; move to the rack
TRIGGER WHEN DISTANCE=1 DELAY=-1 DO Schrittmerker_R1Place(10880,10501,FPlace_R1_L8_S4_VP1,XPlace_R1_L8_S4_VP1) PRIO=-1
;FOLD PTP Place_R1_L8_S4_VP1 CONT Vel=12 % PPlace_R1_L8_S4_VP1 Tool[1]:Upper Gripper Base[0];%{PE}%R8.3.21,%MKUKATPBASIS,%CMOVE,%VPTP,%P 1:PTP, 2:Place_R1_L8_S4_VP1, 3:C_DIS, 5:12, 7:PPlace_R1_L8_S4_VP1
$BWDSTART=FALSE
PDAT_ACT= PPPlace_R1_L8_S4_VP1
FDAT_ACT= FPlace_R1_L8_S4_VP1
BAS(#PTP_PARAMS,12)
PTP XPlace_R1_L8_S4_VP1 C_DIS
;ENDFOLD
TRIGGER WHEN DISTANCE=1 DELAY=-1 DO Schrittmerker_R1Place(10881,10880,FPlace_R1_L8_S4_VP2,XPlace_R1_L8_S4_VP2) PRIO=-1
;FOLD PTP Place_R1_L8_S4_VP2 CONT Vel=12 % PPlace_R1_L8_S4_VP2 Tool[1]:Upper Gripper Base[0];%{PE}%R8.3.21,%MKUKATPBASIS,%CMOVE,%VPTP,%P 1:PTP, 2:Place_R1_L8_S4_VP2, 3:C_DIS, 5:12, 7:PPlace_R1_L8_S4_VP2
$BWDSTART=FALSE
PDAT_ACT= PPPlace_R1_L8_S4_VP2
FDAT_ACT= FPlace_R1_L8_S4_VP2
BAS(#PTP_PARAMS,12)
PTP XPlace_R1_L8_S4_VP2 C_DIS
;ENDFOLD
TRIGGER WHEN DISTANCE=1 DELAY=-1 DO Schrittmerker_R1Place(10882,10881,FPlace_R1_L8_S4_VP3,XPlace_R1_L8_S4_VP3) PRIO=-1
;FOLD PTP Place_R1_L8_S4_VP3 CONT Vel=12 % PPlace_R1_L8_S4_VP3 Tool[1]:Upper Gripper Base[0];%{PE}%R8.3.21,%MKUKATPBASIS,%CMOVE,%VPTP,%P 1:PTP, 2:Place_R1_L8_S4_VP3, 3:C_DIS, 5:12, 7:PPlace_R1_L8_S4_VP3
$BWDSTART=FALSE
PDAT_ACT= PPPlace_R1_L8_S4_VP3
FDAT_ACT= FPlace_R1_L8_S4_VP3
BAS(#PTP_PARAMS,12)
PTP XPlace_R1_L8_S4_VP3 C_DIS
;ENDFOLD
TRIGGER WHEN DISTANCE=1 DELAY=-1 DO Schrittmerker_R1Place(10883,10882,FPlace_R1_L8_S4_VP4,XPlace_R1_L8_S4_VP4) PRIO=-1
;FOLD PTP Place_R1_L8_S4_VP4 CONT Vel=12 % PPlace_R1_L8_S4_VP4 Tool[1]:Upper Gripper Base[0];%{PE}%R8.3.21,%MKUKATPBASIS,%CMOVE,%VPTP,%P 1:PTP, 2:Place_R1_L8_S4_VP4, 3:C_DIS, 5:12, 7:PPlace_R1_L8_S4_VP4
$BWDSTART=FALSE
PDAT_ACT= PPPlace_R1_L8_S4_VP4
FDAT_ACT= FPlace_R1_L8_S4_VP4
BAS(#PTP_PARAMS,12)
PTP XPlace_R1_L8_S4_VP4 C_DIS
;ENDFOLD
TRIGGER WHEN DISTANCE=1 DELAY=-1 DO Schrittmerker_R1Place(10884,10883,FPlace_R1_L8_S4_VP5,XPlace_R1_L8_S4_VP5) PRIO=-1
;FOLD PTP Place_R1_L8_S4_VP5 CONT Vel=12 % PPlace_R1_L8_S4_VP5 Tool[1]:Upper Gripper Base[0];%{PE}%R8.3.21,%MKUKATPBASIS,%CMOVE,%VPTP,%P 1:PTP, 2:Place_R1_L8_S4_VP5, 3:C_DIS, 5:12, 7:PPlace_R1_L8_S4_VP5
$BWDSTART=FALSE
PDAT_ACT= PPPlace_R1_L8_S4_VP5
FDAT_ACT= FPlace_R1_L8_S4_VP5
BAS(#PTP_PARAMS,12)
PTP XPlace_R1_L8_S4_VP5 C_DIS
;ENDFOLD

TRIGGER WHEN DISTANCE=1 DELAY=-1 DO Schrittmerker_R1Place(10885,10884,FPlace_R1_L8_S4_Check,XPlace_R1_L8_S4_Check) PRIO=-1
;FOLD PTP Place_R1_L8_S4_Check Vel=12 % PPlace_R1_L8_S4_Check Tool[1]:Upper Gripper Base[1]:Rack1;%{PE}%R8.3.21,%MKUKATPBASIS,%CMOVE,%VPTP,%P 1:PTP, 2:Place_R1_L8_S4_Check, 3:, 5:12, 7:PPlace_R1_L8_S4_Check
$BWDSTART=FALSE
PDAT_ACT= PPPlace_R1_L8_S4_Check
FDAT_ACT= FPlace_R1_L8_S4_Check
BAS(#PTP_PARAMS,12)
PTP XPlace_R1_L8_S4_Check
;ENDFOLD

;***************************************************
;FOLD Pruefe Platz frei
IF (DetectPart(CHECK_SHELF,PLACE)==OCCUPIED) THEN
  UP_Rueckzug_R1Place( )
  RETURN
ENDIF
;ENDFOLD
;***************************************************

TRIGGER WHEN DISTANCE=1 DELAY=-1 DO Schrittmerker_R1Place(10886,10885,FPlace_R1_L8_S4_VP6,XPlace_R1_L8_S4_VP6) PRIO=-1
;FOLD LIN Place_R1_L8_S4_VP6 CONT Vel=0.5 m/s LPlace_R1_L8_S4_VP6 Tool[1]:Upper Gripper Base[1]:Rack1;%{PE}%R8.3.21,%MKUKATPBASIS,%CMOVE,%VLIN,%P 1:LIN, 2:Place_R1_L8_S4_VP6, 3:C_DIS C_DIS, 5:0.5, 7:LPlace_R1_L8_S4_VP6
$BWDSTART=FALSE
LDAT_ACT= LLPlace_R1_L8_S4_VP6
FDAT_ACT= FPlace_R1_L8_S4_VP6
BAS(#CP_PARAMS,0.5)
LIN XPlace_R1_L8_S4_VP6 C_DIS C_DIS
;ENDFOLD

;FOLD Test the way back home - part 1
CONTINUE
IF ($FLAG[M_Test_GrdstFahren1] AND NOT $FLAG[M_Test_GrdstFahren2]) THEN
  $FLAG[M_Test_GrdstFahren2]=TRUE
  UP_Rueckzug( )
  RETURN
ENDIF
;ENDFOLD

;-------------------------------
; Place part position
;-------------------------------
TRIGGER WHEN DISTANCE=1 DELAY=-1 DO Schrittmerker_R1Place(10887,10888,FPlace_R1_L8_S4_AP,XPlace_R1_L8_S4_AP) PRIO=-1
;FOLD LIN Place_R1_L8_S4_AP Vel=0.2 m/s LPlace_R1_L8_S4_AP Tool[1]:Upper Gripper Base[1]:Rack1;%{PE}%R8.3.21,%MKUKATPBASIS,%CMOVE,%VLIN,%P 1:LIN, 2:Place_R1_L8_S4_AP, 3:, 5:0.2, 7:LPlace_R1_L8_S4_AP
$BWDSTART=FALSE
LDAT_ACT= LLPlace_R1_L8_S4_AP
FDAT_ACT= FPlace_R1_L8_S4_AP
BAS(#CP_PARAMS,0.2)
LIN XPlace_R1_L8_S4_AP
;ENDFOLD

;FOLD Test the way back home - part 2
CONTINUE
IF $FLAG[M_Test_GrdstFahren2] THEN
  $FLAG[M_Test_GrdstFahren2]=FALSE
  UP_Rueckzug( )
  RETURN
ENDIF
;ENDFOLD

;***************************************************
; Disable part lost detection
SetPartLostDetection(NO_PART)
;***************************************************

TRIGGER WHEN DISTANCE=1 DELAY=-1 DO Schrittmerker_R1Place(10888,10889,FPlace_R1_L8_S4_NP1,XPlace_R1_L8_S4_NP1) PRIO=-1
;FOLD LIN Place_R1_L8_S4_NP1 Vel=0.2 m/s LPlace_R1_L8_S4_NP1 Tool[1]:Upper Gripper Base[1]:Rack1;%{PE}%R8.3.21,%MKUKATPBASIS,%CMOVE,%VLIN,%P 1:LIN, 2:Place_R1_L8_S4_NP1, 3:C_DIS C_DIS, 5:0.2, 7:LPlace_R1_L8_S4_NP1
$BWDSTART=FALSE
LDAT_ACT= LLPlace_R1_L8_S4_NP1
FDAT_ACT= FPlace_R1_L8_S4_NP1
BAS(#CP_PARAMS,0.2)
LIN XPlace_R1_L8_S4_NP1
;ENDFOLD

;***************************************************
; Check for part present (empty gripper)
CheckPartPresent(EMPTY_GRIPPER)
;***************************************************
; set load data
SetLoadData( )
;***************************************************

TRIGGER WHEN DISTANCE=1 DELAY=-1 DO Schrittmerker_R1Place(10889,10890,FPlace_R1_L8_S4_NP2,XPlace_R1_L8_S4_NP2) PRIO=-1
;FOLD LIN Place_R1_L8_S4_NP2 Vel=0.5 m/s LPlace_R1_L8_S4_NP2 Tool[1]:Upper Gripper Base[1]:Rack1;%{PE}%R8.3.21,%MKUKATPBASIS,%CMOVE,%VLIN,%P 1:LIN, 2:Place_R1_L8_S4_NP2, 3:, 5:0.5, 7:LPlace_R1_L8_S4_NP2
$BWDSTART=FALSE
LDAT_ACT= LLPlace_R1_L8_S4_NP2
FDAT_ACT= FPlace_R1_L8_S4_NP2
BAS(#CP_PARAMS,0.5)
LIN XPlace_R1_L8_S4_NP2
;ENDFOLD
TRIGGER WHEN DISTANCE=1 DELAY=-1 DO Schrittmerker_R1Place(10890,10891,FPlace_R1_L8_S4_NP3,XPlace_R1_L8_S4_NP3) PRIO=-1
;FOLD PTP Place_R1_L8_S4_NP3 CONT Vel=100 % PPlace_R1_L8_S4_NP3 Tool[1]:Upper Gripper Base[0];%{PE}%R8.3.21,%MKUKATPBASIS,%CMOVE,%VPTP,%P 1:PTP, 2:Place_R1_L8_S4_NP3, 3:C_DIS, 5:100, 7:PPlace_R1_L8_S4_NP3
$BWDSTART=FALSE
PDAT_ACT= PPPlace_R1_L8_S4_NP3
FDAT_ACT= FPlace_R1_L8_S4_NP3
BAS(#PTP_PARAMS,100)
PTP XPlace_R1_L8_S4_NP3 C_DIS
;ENDFOLD
TRIGGER WHEN DISTANCE=1 DELAY=-1 DO Schrittmerker_R1Place(10891,10892,FPlace_R1_L8_S4_NP4,XPlace_R1_L8_S4_NP4) PRIO=-1
;FOLD PTP Place_R1_L8_S4_NP4 CONT Vel=100 % PPlace_R1_L8_S4_NP4 Tool[1]:Upper Gripper Base[0];%{PE}%R8.3.21,%MKUKATPBASIS,%CMOVE,%VPTP,%P 1:PTP, 2:Place_R1_L8_S4_NP4, 3:C_DIS, 5:100, 7:PPlace_R1_L8_S4_NP4
$BWDSTART=FALSE
PDAT_ACT= PPPlace_R1_L8_S4_NP4
FDAT_ACT= FPlace_R1_L8_S4_NP4
BAS(#PTP_PARAMS,100)
PTP XPlace_R1_L8_S4_NP4 C_DIS
;ENDFOLD

TRIGGER WHEN DISTANCE=1 DELAY=-1 DO Schrittmerker_R1Place(10892,10501,FHOME,$nullframe,XHOME) PRIO=-1
;FOLD PTP HOME Vel=100 % PHome;%{PE}%R8.3.21,%MKUKATPBASIS,%CMOVE,%VPTP,%P 1:PTP, 2:HOME, 3:, 5:100, 7:PHome
$BWDSTART=FALSE
PDAT_ACT= PPHome
FDAT_ACT= FHOME
BAS(#PTP_PARAMS,100)
PTP XHOME
;ENDFOLD

;***************************************************
;FOLD Final tasks.
; Robot out of area Rack 1 Level 8
RobAusStorage1_8_A74=RESET_IN_AREA
;***************************************************
; stop cyclic clearence check
$CYCFLAG[ciFreigabeSPS]=DISABLE_MONITORING
;***************************************************
; Disable collision detection
;FOLD COLLDETECT Off ;%{PE}
;FOLD Parameters ;%{h}
;Params IlfProvider=kukaroboter.basistech.inlineforms.colldetect.off; CollDetect.Command=Off
;ENDFOLD
USE_CD_PARAMS(0)
;ENDFOLD
;***************************************************
;ENDFOLD
;***************************************************

END

;###################################################

GLOBAL Def Schrittmerker_R1Place(iMyActPosNo:IN,iMyNextPosNo:IN,fdatMyFDAT:IN,posMyE6POS:IN,axisMyE6AXIS:IN)
INT iMyActPosNo
INT iMyNextPosNo
DECL FDAT fdatMyFDAT
E6POS posMyE6POS
E6AXIS axisMyE6AXIS

iActPosNo = iMyActPosNo
iMyActPosNo = iMyActPosNo - R1_PLACE

CONTINUE
IF NOT(VARSTATE("axisMyE6AXIS") == #INITIALIZED) THEN
  axisMyE6AXIS = {A1 999,A2 999,A3 999,A4 999,A5 999,A6 999,E1 999,E2 999,E3 999,E4 999,E5 999,E6 999}
ENDIF

posRueckzugE6POS[iMyActPosNo] = posMyE6POS
axisRueckzugE6AXIS[iMyActPosNo] = axisMyE6AXIS
iBaseNo[iMyActPosNo] = fdatMyFDAT.BASE_NO
iToolNo[iMyActPosNo] = fdatMyFDAT.TOOL_NO
iNextPosNo[iMyActPosNo] = iMyNextPosNo

CONTINUE
IF ($MOVE_STATE == #PTP_SINGLE) OR ($MOVE_STATE == #PTP_AP01) OR ($MOVE_STATE == #PTP_AP02) THEN
  iMoveTyp[iMyActPosNo]=ciMovePTP
ELSE
  CONTINUE
  IF ($MOVE_STATE == #LIN_SINGLE) OR ($MOVE_STATE == #LIN_AP01) OR ($MOVE_STATE == #LIN_AP02) THEN
    iMoveTyp[iMyActPosNo] = ciMoveLIN
  ELSE
    iMoveTyp[iMyActPosNo] = ciMoveNull
  ENDIF ;($MOVE_STATE==LIN_SINGLE) OR ($MOVE_STATE==LIN_AP01) OR ($MOVE_STATE==LIN_AP02)
ENDIF ;($MOVE_STATE==PTP_SINGLE) OR ($MOVE_STATE==PTP_AP01) OR ($MOVE_STATE==PTP_AP02)

END ;Schrittmerker

;###################################################

GLOBAL DEF UP_Rueckzug_R1Place( )

INT iMyRichtung
INT iMyBereich
INT iMyBereichEnd
INT iMyActPosNo

IRQ4_GND_UP_OFF( )
IRQ5_GND_HP_OFF( )
ZurGrundstFahren_A50=TRUE

iMyBereich = R1_PLACE
iMyBereichEnd = R1_PLACE_END
iMyActPosNo = iActPosNo - iMyBereich

;***************************************************
; Move forewards or backwards?
; Vorwaerts oder rueckwerts fahren?
IF iNextPosNo[iMyActPosNo] > (iActPosNo) THEN
  iMyActPosNo = iNextPosNo[iMyActPosNo] - iMyBereich
  iMyRichtung = ciForward
ELSE
  iMyRichtung = ciBackwards
ENDIF
;***************************************************

REPEAT
  IF (iActPosNo < iMyBereich) OR (iActPosNo > iMyBereichEnd) THEN
    ;***********************************************
    ;          Position ungueltig
    ;  Roboter in T1 in Grundstellung fahren
    ;      Fehler bei Grundstellungsfahrt
    ;        Unbekannter Schrittzaehler
    ErrorHandler(30,#Stoerung)
    ;***********************************************
  ENDIF

  ;*************************************************
  ; Set part lost detection
  ; Check for part present
  SWITCH iActPosNo
  CASE 10013,10034,10054,10074,10095,10120,10137,10158,10178,10197,10218,10238,10261,10278,10297,10316
    SetPartLostDetection(NO_PART)
  CASE 10014,10035,10055,10075,10096,10121,10138,10159,10179,10198,10219,10239,10262,10279,10298,10317
    CheckPartPresent(EMPTY_GRIPPER)
  CASE 10522,10553,10577,10596,10622,10652,10676,10696,10722,10753,10779,10807,10830,10849,10869,10887
    SetPartLostDetection(NO_PART)
  CASE 10523,10554,10578,10597,10623,10653,10677,10697,10723,10754,10780,10808,10831,10850,10870,10888
    CheckPartPresent(EMPTY_GRIPPER)
  ENDSWITCH
  ;*************************************************

  UP_Rueckzug_MoveParam( )

  IF (axisRueckzugE6AXIS[iMyActPosNo].A1 <= $SOFTP_END[1]) THEN
    ;***********************************************
    ; Position is a E6AXIS
    PTP axisRueckzugE6AXIS[iMyActPosNo]
    ;***********************************************
  ELSE
    ;***********************************************
    ; Position is a E6POS
    ;***********************************************
    ; Tool/Base setzen
    IF (iToolNo[iMyActPosNo] == 0) THEN
      $TOOL = $nullframe
    ELSE
      $TOOL = TOOL_DATA[iToolNo[iMyActPosNo]]
    ENDIF
    IF (iBaseNo[iMyActPosNo] == 0) THEN
      $BASE = $nullframe
    ELSE
      $BASE = BASE_DATA[iBaseNo[iMyActPosNo]]
    ENDIF
    ;***********************************************
    ; LIN oder PTP fahren
    ; Koordinaten 0, 0, 0, 0, 0, 0 gelten als ungueltig
    IF (posRueckzugE6POS[iMyActPosNo].x == 0) AND (posRueckzugE6POS[iMyActPosNo].y == 0) AND (posRueckzugE6POS[iMyActPosNo].z == 0) AND (posRueckzugE6POS[iMyActPosNo].a == 0) AND (posRueckzugE6POS[iMyActPosNo].b == 0) AND (posRueckzugE6POS[iMyActPosNo].c == 0) THEN
      ErrorHandler(30,#STOERUNG)
    ENDIF
    SWITCH iMoveTyp[iMyActPosNo + iMyRichtung]
    CASE ciMoveLIN
      LIN posRueckzugE6POS[iMyActPosNo]
    CASE ciMovePTP
      PTP posRueckzugE6POS[iMyActPosNo]
    DEFAULT
      PTP posRueckzugE6POS[iMyActPosNo]
    ENDSWITCH
    ;***********************************************
  ENDIF

  ;*************************************************
  ; Set next position
  WAIT SEC 0
  iActPosNo = iNextPosNo[iMyActPosNo]
  iMyActPosNo = iActPosNo - iMyBereich
  ;*************************************************

UNTIL $IN_HOME OR $IN_HOME1

ZurGrundstFahren_A50=FALSE

;***************************************************
; Disable collision detection
;FOLD COLLDETECT Off ;%{PE}
;FOLD Parameters ;%{h}
;Params IlfProvider=kukaroboter.basistech.inlineforms.colldetect.off; CollDetect.Command=Off
;ENDFOLD
USE_CD_PARAMS(0)
;ENDFOLD
;***************************************************

AnfStoer_Store1_1_A99=RESET_REQUEST
AnfStoer_Store1_2_A100=RESET_REQUEST
AnfStoer_Store1_3_A101=RESET_REQUEST
AnfStoer_Store1_4_A102=RESET_REQUEST
AnfStoer_Store1_5_A103=RESET_REQUEST
AnfStoer_Store1_6_A104=RESET_REQUEST
AnfStoer_Store1_7_A105=RESET_REQUEST
AnfStoer_Store1_8_A106=RESET_REQUEST

RobAusStorage1_1_A67=RESET_IN_AREA
RobAusStorage1_2_A68=RESET_IN_AREA
RobAusStorage1_3_A69=RESET_IN_AREA
RobAusStorage1_4_A70=RESET_IN_AREA
RobAusStorage1_5_A71=RESET_IN_AREA
RobAusStorage1_6_A72=RESET_IN_AREA
RobAusStorage1_7_A73=RESET_IN_AREA
RobAusStorage1_8_A74=RESET_IN_AREA

$CYCFLAG[ciFreigabeSPS]=DISABLE_MONITORING

WAIT SEC 0

END ; UP_Rueckzug_R1Place( )
